FUNCTION_BLOCK HRL_OperatingModes
VAR_INPUT
	Start 			: BOOL;
	Stop			: BOOL;
	Reset			: BOOL;
	Schalter		: BOOL;
	Schrittkette_GS	: BOOL;
	Count1 : INT := 0;
	Count2 : INT := 0;
	Alt_abort: BOOL;
	Err_detected: BOOL;
	Diag_finished: BOOL;
	Alt_found: BOOL;
	Cycle_finished: BOOL;

END_VAR
VAR_OUTPUT
	{attribute 'OPC.UA.DA' := '1'} // für OPC UA freigeben
	A1 : BOOL := FALSE; //Initialzustand
	{attribute 'OPC.UA.DA' := '1'} // für OPC UA freigeben
	A2 : BOOL; //Stillstand angefordert am Ende des Zyklus
//	A3 : BOOL; //Stillstand angefordert in einem bestimmten Zustand
//	A4 : BOOL; //Erhaltener Stillstand
	{attribute 'OPC.UA.DA' := '1'} // für OPC UA freigeben
	A5 : BOOL; //Vorbereitung zur Wiederaufnahme nach Störung
	{attribute 'OPC.UA.DA' := '1'} // für OPC UA freigeben
	A6 : BOOL; //Fahrt in den Initialzustand
	{attribute 'OPC.UA.DA' := '1'} // für OPC UA freigeben
	F1 : BOOL; //Normalbetrieb
//	F2 : BOOL; //Anfahren
//	F3 : BOOL; //Abfahren
	{attribute 'OPC.UA.DA' := '1'} // für OPC UA freigeben
	F4 : BOOL; //Handbetrieb
//	F5 : BOOL; //Schrittbetrieb
//	F6 : BOOL; //Testbetrieb
	{attribute 'OPC.UA.DA' := '1'} // für OPC UA freigeben
	D1 : BOOL; //Not-Aus
	{attribute 'OPC.UA.DA' := '1'} // für OPC UA freigeben
	D2 : BOOL; //Diagnose und Störbehandlung
	{attribute 'OPC.UA.DA' := '1'} // für OPC UA freigeben
	D3 : BOOL; //Produktion trotz Störung
	MethodCall_InitStateDrive : BOOL;
	InputVar_InitStateDrive : BOOL;
END_VAR
VAR
	bFirstScan : BOOL := TRUE;
	FirstScanCount: INT := 0;
	AlwaysTrue : BOOL := TRUE;
	TestingVariable : BOOL;	
	 nTaskIdx : DINT;
	RS_InitialState: RS;
	RS_InitialState11: RS;	
	RS_InitialDrive: RS;
	RS_ManualOperationMode: RS;
	RS_AutomaticOperationMode: RS;
	RS_CycleEnded: RS;
	//Count: INT := 0;
	R_TRIG_Manual: R_TRIG;
	R_TRIG_Automatic: R_TRIG;
	R_TRIG_InitialDrive: R_TRIG;
	R_TRIG_CycleEnded: R_TRIG;
	R_TRIG_Init: R_TRIG;
	NeverTrue: BOOL := FALSE;
	SR_D1: SR;
	RS_D2: RS;
	
	RS_D3: RS;
	RS_A5: RS;
	
	
	bFirstCycle: BOOL;
END_VAR
VAR // added by the converter: edge detectors and wires of the graphical bodies
    _w1, _w2, _w3, _w4 : BOOL;
END_VAR

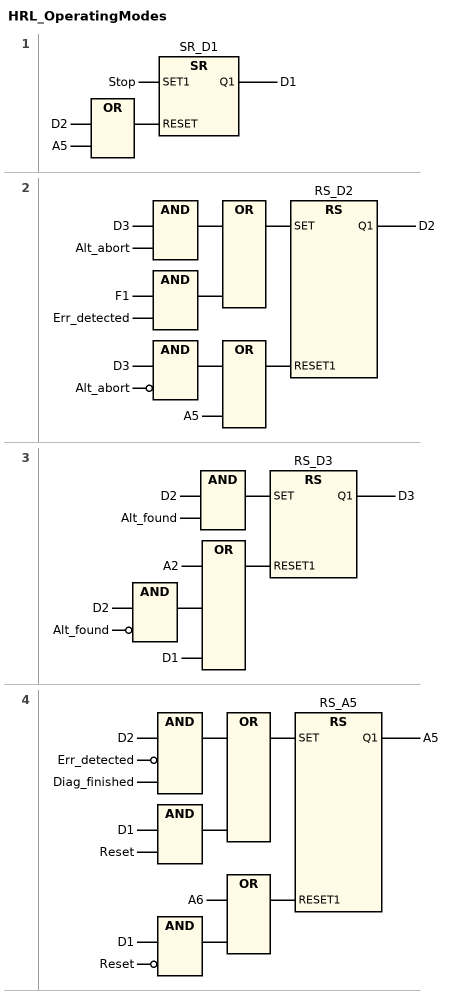
// NETWORK 1
SR_D1(SET1 := Stop, RESET := D2 OR A5); // SR
D1 := SR_D1.Q1;

// NETWORK 2
RS_D2(SET := D3 AND Alt_abort OR F1 AND Err_detected, RESET1 := D3 AND NOT Alt_abort OR A5); // RS
D2 := RS_D2.Q1;

// NETWORK 3
RS_D3(SET := D2 AND Alt_found, RESET1 := A2 OR D2 AND NOT Alt_found OR D1); // RS
D3 := RS_D3.Q1;

// NETWORK 4
RS_A5(SET := D2 AND NOT Err_detected AND Diag_finished OR D1 AND Reset, RESET1 := A6 OR D1 AND NOT Reset); // RS
A5 := RS_A5.Q1;

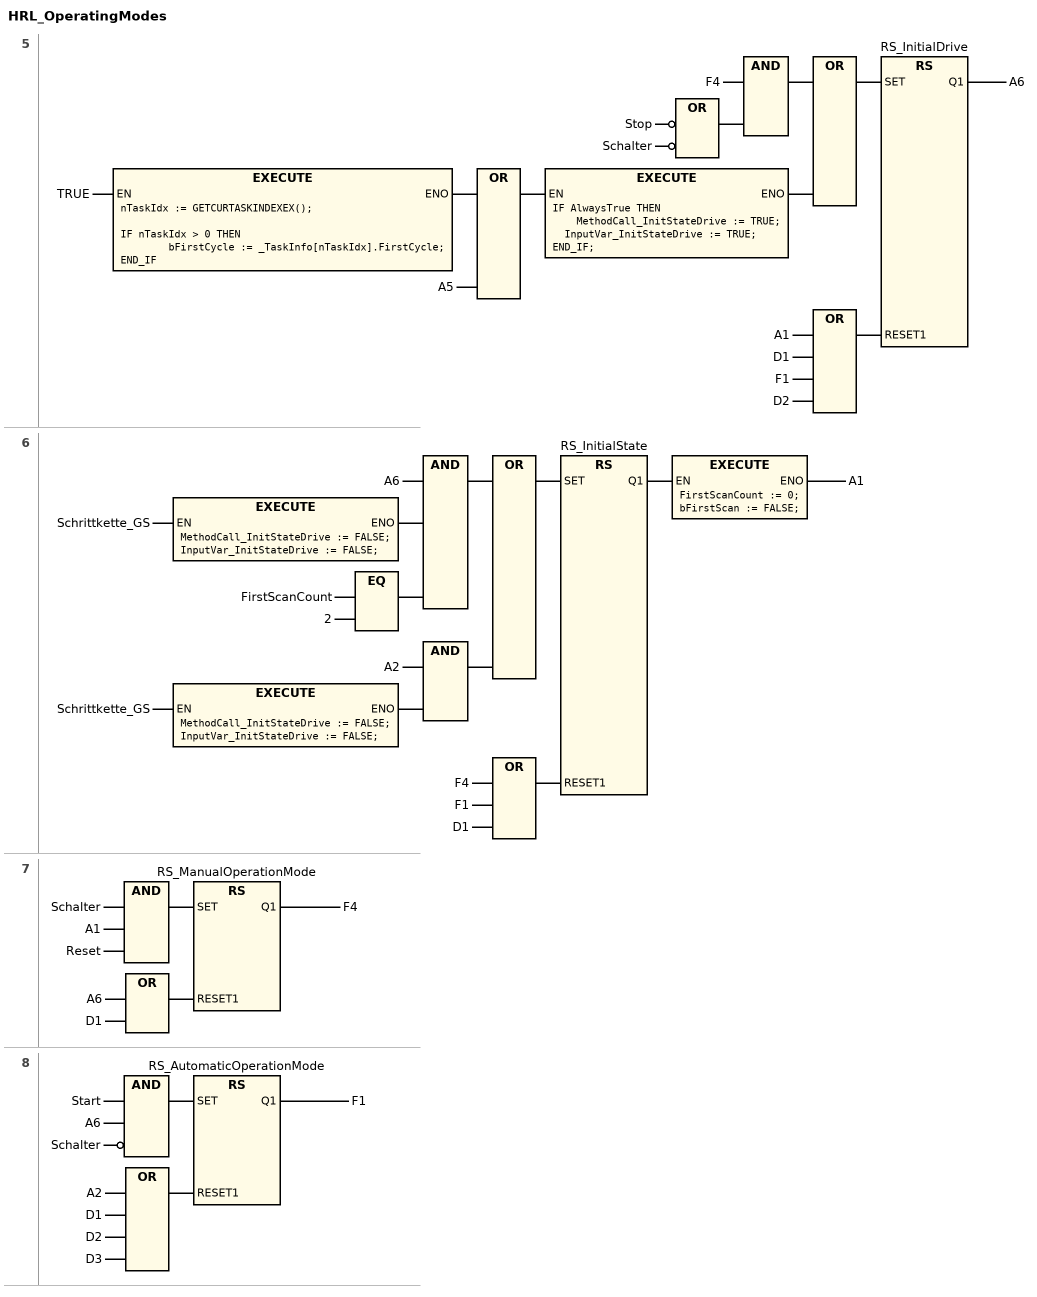
// NETWORK 5
nTaskIdx := GETCURTASKINDEXEX();

IF nTaskIdx > 0 THEN
        bFirstCycle := _TaskInfo[nTaskIdx].FirstCycle;
END_IF
_w1 := TRUE OR A5;
IF _w1 THEN
    IF AlwaysTrue THEN
        MethodCall_InitStateDrive := TRUE;
    	InputVar_InitStateDrive := TRUE;
    END_IF;
END_IF
RS_InitialDrive(SET := F4 AND (NOT Stop OR NOT Schalter) OR _w1, RESET1 := A1 OR D1 OR F1 OR D2); // RS
A6 := RS_InitialDrive.Q1;

// NETWORK 6
_w2 := Schrittkette_GS;
IF _w2 THEN
    MethodCall_InitStateDrive := FALSE;
    InputVar_InitStateDrive := FALSE;
END_IF
_w3 := Schrittkette_GS;
IF _w3 THEN
    MethodCall_InitStateDrive := FALSE;
    InputVar_InitStateDrive := FALSE;
END_IF
RS_InitialState(SET := A6 AND _w2 AND FirstScanCount = 2 OR A2 AND _w3, RESET1 := F4 OR F1 OR D1); // RS
_w4 := RS_InitialState.Q1;
IF _w4 THEN
    FirstScanCount := 0;
    bFirstScan := FALSE;
END_IF
A1 := _w4;

// NETWORK 7
RS_ManualOperationMode(SET := Schalter AND A1 AND Reset, RESET1 := A6 OR D1); // RS
F4 := RS_ManualOperationMode.Q1;

// NETWORK 8
RS_AutomaticOperationMode(SET := Start AND A6 AND NOT Schalter, RESET1 := A2 OR D1 OR D2 OR D3); // RS
F1 := RS_AutomaticOperationMode.Q1;

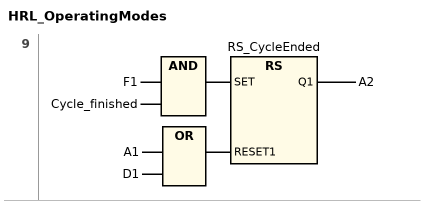
// NETWORK 9
RS_CycleEnded(SET := F1 AND Cycle_finished, RESET1 := A1 OR D1); // RS
A2 := RS_CycleEnded.Q1;

END_FUNCTION_BLOCK

(* stored: Version 1.1.0.1, ProductVersion 3.1.4026.18
   POU HRL_OperatingModes: Id {cdeda4f8-1e28-4a09-b37b-b8311b19316e}, SpecialFunc None *)
